# EPICS IOC start-up script: Keithley/iocBoot/iocKeith6430/cool.iocsh
epicsEnvSet "STREAM_PROTOCOL_PATH", "$(TOP)"

drvAsynIPPortConfigure "$(PORT)", "localhost:5555"

dbLoadRecords("$(TOP)/db/stream.db" "P=$(user):,PORT=$(PORT)")
